(* IEC 61131-3 sources: ST-to-Python-Transpiler/AS Projekti/MySignalTools/Program, 3 files *)

(* ---- Types.typ ---- *)
TYPE

END_TYPE

(* ---- SignalProcess.st ---- *)
PROGRAM _INIT
	(* Insert code here *)

END_PROGRAM

PROGRAM _CYCLIC
	LimiterFB(IN := AnalogRaw, MIN_LIMIT := -10.0, MAX_LIMIT := 10.0, HYSTERESIS := 0.2);
	LimiterFB();

	LimitedSignal := LimiterFB.OUT;

	DebounceFB(TRIG := ButtonInput, DEBOUNCE_CYCLES := 20);
	DebounceFB();

	IF DebounceFB.VALID_EDGE THEN
		IntegratorEnabled := NOT IntegratorEnabled;
	END_IF;

	IntegratorFB(IN := LimitedSignal, DT_STEP := 0.01, ENABLE := IntegratorEnabled, RESET := FALSE, MAX_ACCUM := 100.0, DELTA_LIMIT := 0.5);
	IntegratorFB();

	AccumulatedResult := IntegratorFB.OUT;

END_PROGRAM

PROGRAM _EXIT
	(* Insert code here *)

END_PROGRAM

(* ---- Variables.var ---- *)
VAR
	AnalogRaw : REAL := 12.3;         (** Noisy sensor input signal **)
	ButtonInput : BOOL := FALSE;     (** Digital input to toggle signal integration **)

	AccumulatedResult : REAL;        (** Result of signal integration **)
	LimitedSignal : REAL;            (** Signal after limiting/clamping **)
	IntegratorEnabled : BOOL;        (** Indicates if integration is currently active **)

	LimiterFB : SignalLimiter;
	DebounceFB : ToggleDebounce;
	IntegratorFB : SignalIntegrator;

END_VAR

VAR CONSTANT

END_VAR
